FUNCTION F_ROUND_REAL : LREAL
VAR_INPUT
	rInput : LREAL;
  	iDecimalPlaces : INT;
END_VAR
VAR
	rFactor : LREAL;
    rScaled : LREAL;
    rRounded : LREAL;
END_VAR

rFactor := EXPT(10.0, iDecimalPlaces);         // Ex: 100.0 for 2 digits
rScaled := rInput * rFactor;

IF rScaled >= 0.0 THEN
    rRounded := TRUNC(rScaled + 0.5);
ELSE
    rRounded := TRUNC(rScaled - 0.5);
END_IF

F_ROUND_REAL := rRounded / rFactor;

END_FUNCTION

(* stored: Version 1.1.0.1, ProductVersion 3.1.4024.12
   POU F_ROUND_REAL: Id {95848e51-29c9-47b8-ba91-f91034e23531}, SpecialFunc None *)
